# EPICS substitutions: BLDApp/Db/fcom_stats.substitutions
#
# FCOM statistics substitutions file
# Add one entry for each FCOM blob
# Index numbers and BLOB names must match bldPulseBlobs array in BLDMCast.c
#

file fcom_stats.template
{
	pattern
	{	NUM,	BLOB		}
	{	0,		"TMIT"		}
	{	1,		"ENG1"		}
	{	2,		"ENG2"		}
	{	3,		"POS1"		}
	{	4,		"POS2"		}
	{	5,		"POS3"		}
	{	6,		"POS4"		}
# TODO: Rename BLEN to BC2CH here and in BLDMCast.c
	{	7,		"BLEN"		}
	{	8,		"BC2EN"		}
	{	9,		"BC1CH"		}
	{	10,		"BC1EN"		}
	{	11,		"UND"		}
	{	12,		"DMP_CHARGE"}
	{	13,		"XTCAV_AMP"	}
# LTU States from FastFeedback. This replaces POS{1,2,3,4} above.
    {   14,     "LTU"       }
}
